{attribute 'linkalways'} 
{attribute 'no_explicit_call' := 'This FB is a CLASS and must be accessed using methods or properties'}
{attribute 'enable_dynamic_creation'}
FUNCTION_BLOCK _Array0to6OfLREAL EXTENDS ArrayDatatypeBase_1D
VAR CONSTANT
	lBound : DINT := 0;
	uBound : DINT := 6;
END_VAR
VAR
	localData : ARRAY [lBound..uBound] OF LREAL;
	activeData : REFERENCE TO ARRAY [lBound..uBound] OF LREAL REF= localData;
	elements : ARRAY [lBound..uBound] OF _LREAL(0.0);
	baseType : _LREAL(0.0);
END_VAR

PROPERTY PUBLIC Address : PVOID
GET
Address := ADR(activeData);
END_GET
END_PROPERTY

PROPERTY PUBLIC BaseDatatype : I_Datatype
GET
BaseDatatype := baseType;
END_GET
END_PROPERTY

METHOD PUBLIC ClearReference
VAR_INPUT
END_VAR
activeData REF= localData;
SetElementReference();
END_METHOD

METHOD PUBLIC Clone : I_Datatype
VAR
    pClone : POINTER TO _Array0to6OfLREAL;
END_VAR
pClone := __NEW(_Array0to6OfLREAL());
pClone^.Value := Value;
Clone := pClone^;
END_METHOD

METHOD FB_init : BOOL
VAR_INPUT
	bInitRetains : BOOL; // if TRUE, the retain variables are initialized (warm start / cold start)
	bInCopyCode : BOOL;  // if TRUE, the instance afterwards gets moved into the copy code (online change)
END_VAR
SetElementReference();
END_METHOD

METHOD PUBLIC MakeReferenceTo
VAR_INPUT
	ReferenceTarget : REFERENCE TO ARRAY [lBound..uBound] OF LREAL;
END_VAR
activeData REF= ReferenceTarget;
SetElementReference();
END_METHOD

METHOD PROTECTED OnSerializeArrayValues
VAR_INPUT
	Serializer : I_Serializer;
END_VAR
VAR
	i : DINT;
END_VAR
FOR i := lBound TO uBound DO
	elements[i].SerializeWith(Serializer);
END_FOR
END_METHOD

METHOD PROTECTED SetElementReference
VAR_INPUT
END_VAR
VAR
	i : DINT;
END_VAR
FOR i := lBound TO uBound DO
	elements[i].MakeReferenceTo(activeData[i]);
END_FOR
END_METHOD

PROPERTY PUBLIC Size : UDINT
GET
Size := SIZEOF(activeData);
END_GET
END_PROPERTY

METHOD PROTECTED TryDeserializeArrayValues : BOOL
VAR_INPUT
	Deserializer : I_Deserializer;
	Feedback : I_DeserializerFeedback;
END_VAR
VAR
	enumerator : I_DeserializerArrayForwardEnumerator;
	i : DINT;
END_VAR
enumerator := Deserializer.GetArrayEnumerator();
i := lBound;

WHILE enumerator.MoveNext() AND i <= uBound DO
	
	IF NOT elements[i].TryDeserializeFrom(enumerator.Current, Feedback) THEN
		EXIT;
	END_IF
	i := i + 1;

END_WHILE
enumerator.Dispose();
END_METHOD

METHOD PUBLIC TryGetElementAsDatatypeByIndex : BOOL
VAR_INPUT
	Index : DINT;
	Destination : REFERENCE TO I_Datatype;
END_VAR
IF Index < lbound OR Index > ubound THEN
	RETURN;
END_IF

Destination := elements[Index];
TryGetElementAsDatatypeByIndex := TRUE;
END_METHOD

METHOD PUBLIC TryGetLowerBound : BOOL
VAR_INPUT
	Dimention : UDINT;
	Destination : REFERENCE TO DINT;
END_VAR
IF Dimention = 1 THEN
	Destination := lBound;
	TryGetLowerBound := TRUE;
END_IF
END_METHOD

METHOD PUBLIC TryGetUpperBound : BOOL
VAR_INPUT
	Dimention : UDINT;
	Destination : REFERENCE TO DINT;
END_VAR
IF Dimention = 1 THEN
	Destination := uBound;
	TryGetUpperBound := TRUE;
END_IF
END_METHOD

METHOD TryMakeReferenceTo : BOOL
VAR_INPUT
	Target : I_Datatype;
END_VAR
VAR
	pTargetData : POINTER TO ARRAY [lBound..uBound] OF LREAL;
END_VAR
IF NOT IsEquivalentTo(Target) THEN
	RETURN;
END_IF

pTargetData := Target.Address;
activeData REF= pTargetData^;
SetElementReference();
TryMakeReferenceTo := TRUE;
END_METHOD

PROPERTY PUBLIC Value : REFERENCE TO ARRAY [lBound..uBound] OF LREAL;
GET
Value ref= activeData;
END_GET
END_PROPERTY

END_FUNCTION_BLOCK

(* stored: Version 1.1.0.1, ProductVersion 3.1.4024.13
   POU _Array0to6OfLREAL: Id {1c20c713-00d9-0e5d-12c2-b9891e49dda2}, SpecialFunc None
   Folder Core: Id {8165bb38-1db7-09a0-34a3-e6381faa7325}
   Folder Constructor: Id {50f70370-37f9-0c00-35ce-2c5c2f265c3e}
   Folder Protected: Id {2af376a5-bf63-0ad5-005b-bc3aacd9394d}
   Folder Customize: Id {b1e8b6c5-d330-00ae-37db-2e9ebfaa01db}
   Property Address: Id {3e4e8bd7-df2e-00f3-0bbe-e39720e88c93}
   Get Get: Id {966ccad1-802f-06c2-2b11-a6edb8b068d8}
   Property BaseDatatype: Id {ddbbff71-67d6-0d32-3450-8f0143216007}
   Get Get: Id {71266db4-a8f3-020d-11ca-3199d5eb2e31}
   Method ClearReference: Id {d868d69d-2145-0c9b-0247-ddc6b9132fe2}
   Method Clone: Id {190e9f73-95ac-0a35-13f9-1864d9a3ad0b}
   Method FB_init: Id {d319c687-cf2c-02d7-1075-73983eb63726}
   Method MakeReferenceTo: Id {8cc53f04-7d47-0d7e-2edb-6609abfea6ec}
   Method OnSerializeArrayValues: Id {a8a47aae-c7ea-06f4-0452-5af541695ca9}
   Method SetElementReference: Id {02b10f2a-fe62-0058-2571-739f507f78e6}
   Property Size: Id {bca2f301-3447-096e-1d89-64d2459e5540}
   Get Get: Id {385aaf2d-cd41-04a3-319b-f60cce5d34e0}
   Method TryDeserializeArrayValues: Id {a14be4b6-d62d-0f16-211d-5fdeefa1b1ac}
   Method TryGetElementAsDatatypeByIndex: Id {0c08f76b-eed6-0ec8-17a1-4cf5bb0a68d8}
   Method TryGetLowerBound: Id {da3a2da9-8c51-0918-36a1-7520ffbc6782}
   Method TryGetUpperBound: Id {5203dd1d-1790-0e9b-0570-d87107c78189}
   Method TryMakeReferenceTo: Id {57d9a9db-d4cd-0f3c-2d4a-199aa75b9c98}
   Property Value: Id {f29670fc-0b46-0e4a-26d9-1b9a3bfb538b}
   Get Get: Id {866fc21d-b706-0f4d-1bfd-d5f64b98cb70} *)
